// TIA Portal project "正反转流水线控制（核心程序）" (V16)

(* hardware
DEVICE "S7-1200 station_1"  S7-1200 Station
   slot 0: "Rack_0"  S7-1200 Rack  Rack  V1.0
   slot 1: "PLC_1"  CPU 1214C DC/DC/Rly  6ES7 214-1HG40-0XB0  V4.4
DEVICE "HMI_1"  KTP700 Basic PN
   slot 0: "HMI_1"  KTP700 Basic PN  6AV2 123-2GB03-0AX0  16.0.0.0
   slot 1: "HMI_RT_1"  KTP700 Basic PN  6AV2 123-2GB03-0AX0  16.0.0.0
   slot 5: "HMI_1.IE_CP_1"  PROFINET Interface  16.0.0.0
      slot 1: "PROFINET Interface_1"  PROFINET Interface
         slot 1: "Port_1"  Port
*)

// ===== PLC "PLC_1"  CPU 1214C DC/DC/Rly =====

VAR_GLOBAL   // PLC tag table "默认变量表"
   "Tag_1" AT %M20.0 : Bool;
END_VAR

VAR_GLOBAL   // PLC tag table "中间变量"
   "启动(1)" AT %M0.0 : Bool;
   "停止" AT %M0.1 : Bool;
   "复位(1)" AT %M0.2 : Bool;
   "启动标志" AT %M0.3 : Bool;
   "中间寄存器1" AT %MD100 : DInt;
   "收料皮带启动" AT %M0.4 : Bool;
   "中间寄存器2" AT %MD104 : DInt;
   "判断是否" AT %M0.5 : Bool;
   "中间变量1" AT %M0.6 : Bool;
   "中间寄存器3" AT %MD108 : DInt;
   "中间变量2" AT %M0.7 : Bool;
   "中间变量2(1)" AT %M1.0 : Bool;
   "中间变量3" AT %M1.1 : Bool;
END_VAR

VAR_GLOBAL   // PLC tag table "io表"
   "上料端传感器" AT %I2.0 : Bool;
   "中断传感器" AT %I2.1 : Bool;
   "下料传感器" AT %I2.2 : Bool;
   "启动" AT %I2.3 : Bool;
   "复位" AT %I2.4 : Bool;
   "急停" AT %I2.5 : Bool;
   "挡位1" AT %I2.6 : Bool;
   "急停按钮" AT %I2.7 : Bool;
   "FACTORY I/O (Running)" AT %I1.0 : Bool;
   "卡槽" AT %Q2.0 : Bool;
   "绿色" AT %Q2.1 : Bool;
   "黄色" AT %Q2.2 : Bool;
   "红色" AT %Q2.3 : Bool;
   "上料" AT %Q2.4 : Bool;
   "取料" AT %Q2.5 : Bool;
   "速度" AT %ID30 : Real;
   "皮带1" AT %QD30 : Real;
   "皮带2" AT %QD34 : Real;
   "显示屏" AT %QD38 : DInt;
END_VAR

DATA_BLOCK "数据块_1"   // DB1
{ S7_Optimized_Access := 'TRUE' }
VERSION : 0.1
   VAR
      中间变量1 : Bool := 0;
      中间变量2 : Bool := 0;
   END_VAR
BEGIN
END_DATA_BLOCK

FUNCTION "MHJ-PLC-Lab-Function-S71200" : Void   // FC9000, SCL
{ S7_Optimized_Access := 'TRUE' }
VERSION : 0.1
   VAR_TEMP
      rdTimeReturn : Int;
      outputTime : DTL;
      SyncVal : Byte;
      forVal : Int;
      forVal_2 : Int;
      Value : Byte;
   END_VAR
   VAR CONSTANT
      CompVal : Byte := 16#34;
      Value_01 : Byte := 16#11;
      Value_01_DW : DWord := 16#A165_D992;
      Value_02_DW : DWord := 16#58BE_4401;
   END_VAR
BEGIN

   #Value:=PEEK(area := 16#82,
        dbNumber := 0,
        byteOffset := 511);
   #Value := #Value + 1;

   POKE(area := 16#82,
        dbNumber := 0,
        byteOffset := 511,
        value := #Value);

   POKE(area:=16#81,
        dbNumber:=0,
        byteOffset:=1016,
        value:=#Value_01_DW);
   POKE(area := 16#81,
        dbNumber := 0,
        byteOffset := 1020,
        value := #Value_02_DW);

   POKE(area := 16#81,
        dbNumber := 0,
        byteOffset := 511,
        value := B#16#00);

   FOR #forVal := 0 TO 120 DO
       FOR #forVal_2:=0 TO 10 DO
           #rdTimeReturn:=RD_SYS_T(#outputTime);
           #rdTimeReturn := WR_SYS_T(#outputTime);
           #rdTimeReturn := RD_SYS_T(#outputTime);
           #rdTimeReturn := WR_SYS_T(#outputTime);
       END_FOR;
       #SyncVal:= PEEK(area := 16#81,
                      dbNumber := 0,
                      byteOffset := 511);
       IF #SyncVal = #CompVal THEN
          GOTO M_1;
       END_IF;
   END_FOR;
   RETURN;

   M_1:
   POKE(area := 16#81,
        dbNumber := 0,
        byteOffset := 511,
        value := B#16#0);
END_FUNCTION

ORGANIZATION_BLOCK "Main"   // OB1, LAD, ProgramCycle
TITLE = "Main Program Sweep (Cycle)"
{ S7_Optimized_Access := 'TRUE' }
VERSION : 0.1
   VAR_INPUT
      Initial_Call : Bool;   // Initial call of this OB
      Remanence : Bool;   // =True, if remanent data are available
   END_VAR
   VAR_TEMP   // added for the SCL form of the ladder/FBD networks
      _w1 : Bool;
      _w2 : Bool;
   END_VAR
BEGIN

REGION Network 1
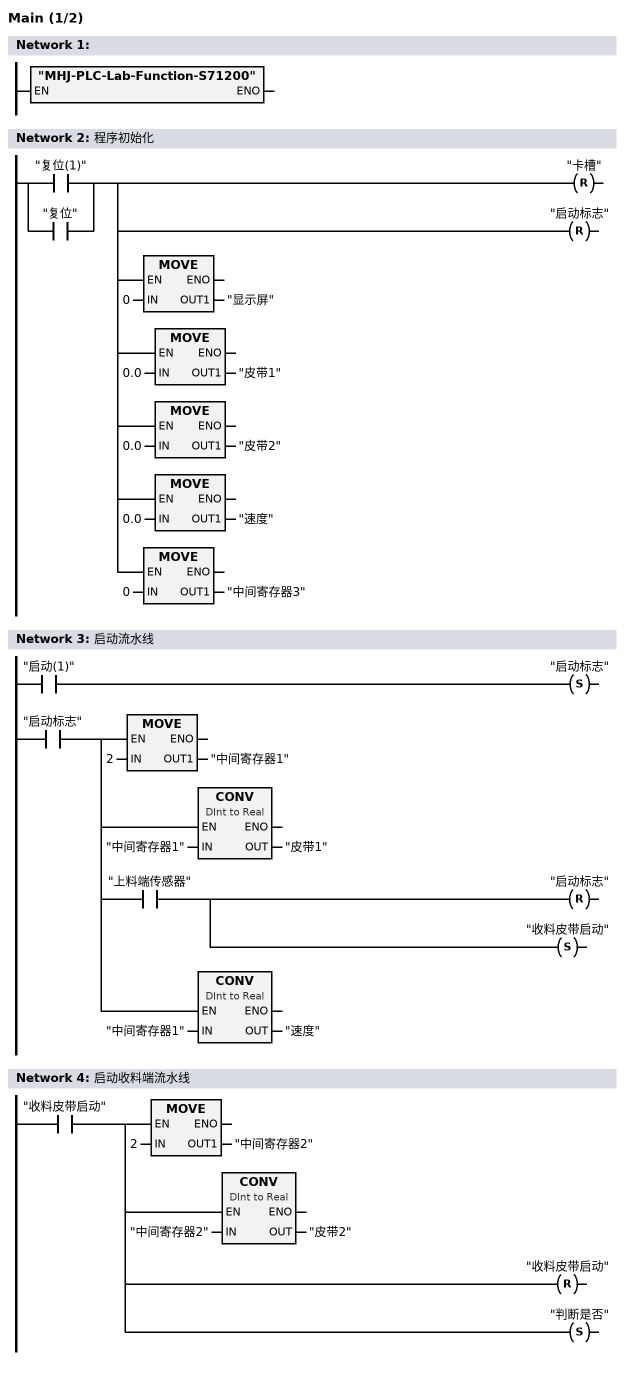
   RUNG wire#powerrail
      "MHJ-PLC-Lab-Function-S71200"()
   END_RUNG
   // the same network as SCL:
   "MHJ-PLC-Lab-Function-S71200"();
END_REGION

REGION Network 2: 程序初始化
   RUNG wire#powerrail
      Contact( "复位(1)" )
      wire#w1
      R_Coil( "卡槽" )
   END_RUNG
   RUNG wire#powerrail
      Contact( "复位" )
   END_RUNG wire#w1
   RUNG wire#w1
      R_Coil( "启动标志" )
   END_RUNG
   RUNG wire#w1
      Move(in := 0, out1 => "显示屏")
   END_RUNG
   RUNG wire#w1
      Move(in := 0.0, out1 => "皮带1")
   END_RUNG
   RUNG wire#w1
      Move(in := 0.0, out1 => "皮带2")
   END_RUNG
   RUNG wire#w1
      Move(in := 0.0, out1 => "速度")
   END_RUNG
   RUNG wire#w1
      Move(in := 0, out1 => "中间寄存器3")
   END_RUNG
   // the same network as SCL:
   IF "复位(1)" OR "复位" THEN
       "卡槽" := FALSE;
       "启动标志" := FALSE;
       "显示屏" := 0;
       "皮带1" := 0.0;
       "皮带2" := 0.0;
       "速度" := 0.0;
       "中间寄存器3" := 0;
   END_IF;
END_REGION

REGION Network 3: 启动流水线
   RUNG wire#powerrail
      Contact( "启动(1)" )
      S_Coil( "启动标志" )
   END_RUNG
   RUNG wire#powerrail
      Contact( "启动标志" )
      wire#w1
      Move(in := 2, out1 => "中间寄存器1")
   END_RUNG
   RUNG wire#w1
      { S7_Templates := "[SrcType := DInt, DestType := Real]" } Convert(in := "中间寄存器1", out => "皮带1")
   END_RUNG
   RUNG wire#w1
      Contact( "上料端传感器" )
      wire#w2
      R_Coil( "启动标志" )
   END_RUNG
   RUNG wire#w2
      S_Coil( "收料皮带启动" )
   END_RUNG
   RUNG wire#w1
      { S7_Templates := "[SrcType := DInt, DestType := Real]" } Convert(in := "中间寄存器1", out => "速度")
   END_RUNG
   // the same network as SCL:
   IF "启动(1)" THEN "启动标志" := TRUE; END_IF;
   IF "启动标志" THEN
       "中间寄存器1" := 2;
       "皮带1" := DINT_TO_REAL("中间寄存器1");
   END_IF;
   #_w1 := "启动标志";
   #_w2 := "启动标志" AND "上料端传感器";
   IF #_w2 THEN
       "启动标志" := FALSE;
       "收料皮带启动" := TRUE;
   END_IF;
   IF #_w1 THEN "速度" := DINT_TO_REAL("中间寄存器1"); END_IF;
END_REGION

REGION Network 4: 启动收料端流水线
   RUNG wire#powerrail
      Contact( "收料皮带启动" )
      wire#w1
      Move(in := 2, out1 => "中间寄存器2")
   END_RUNG
   RUNG wire#w1
      { S7_Templates := "[SrcType := DInt, DestType := Real]" } Convert(in := "中间寄存器2", out => "皮带2")
   END_RUNG
   RUNG wire#w1
      R_Coil( "收料皮带启动" )
   END_RUNG
   RUNG wire#w1
      S_Coil( "判断是否" )
   END_RUNG
   // the same network as SCL:
   IF "收料皮带启动" THEN
       "中间寄存器2" := 2;
       "皮带2" := DINT_TO_REAL("中间寄存器2");
   END_IF;
   #_w1 := "收料皮带启动";
   IF #_w1 THEN
       "收料皮带启动" := FALSE;
       "判断是否" := TRUE;
   END_IF;
END_REGION

REGION Network 5: 计数
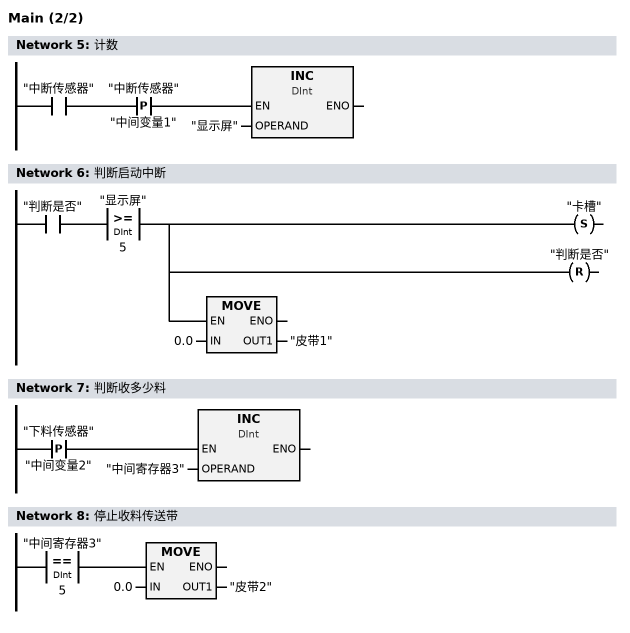
   RUNG wire#powerrail
      Contact( "中断传感器" )
      P_Contact(operand := "中断传感器", bit := "中间变量1")
      { S7_Templates := "DestType := DInt" } Inc( "显示屏" )
   END_RUNG
   // the same network as SCL:
   #_w1 := "中断传感器" AND "中断传感器" AND NOT "中间变量1";   // rising edge of "中断传感器"
   "中间变量1" := "中断传感器";
   IF #_w1 THEN "显示屏" := "显示屏" + 1; END_IF;
END_REGION

REGION Network 6: 判断启动中断
   RUNG wire#powerrail
      Contact( "判断是否" )
      { S7_Templates := "SrcType := DInt" } GE_Contact(in1 := "显示屏", in2 := 5)
      wire#w1
      S_Coil( "卡槽" )
   END_RUNG
   RUNG wire#w1
      R_Coil( "判断是否" )
   END_RUNG
   RUNG wire#w1
      Move(in := 0.0, out1 => "皮带1")
   END_RUNG
   // the same network as SCL:
   IF "判断是否" AND ("显示屏" >= 5) THEN "卡槽" := TRUE; END_IF;
   #_w1 := "判断是否" AND ("显示屏" >= 5);
   IF #_w1 THEN
       "判断是否" := FALSE;
       "皮带1" := 0.0;
   END_IF;
END_REGION

REGION Network 7: 判断收多少料
   RUNG wire#powerrail
      P_Contact(operand := "下料传感器", bit := "中间变量2")
      { S7_Templates := "DestType := DInt" } Inc( "中间寄存器3" )
   END_RUNG
   // the same network as SCL:
   #_w1 := "下料传感器" AND NOT "中间变量2";   // rising edge of "下料传感器"
   "中间变量2" := "下料传感器";
   IF #_w1 THEN "中间寄存器3" := "中间寄存器3" + 1; END_IF;
END_REGION

REGION Network 8: 停止收料传送带
   RUNG wire#powerrail
      { S7_Templates := "SrcType := DInt" } EQ_Contact(in1 := "中间寄存器3", in2 := 5)
      Move(in := 0.0, out1 => "皮带2")
   END_RUNG
   // the same network as SCL:
   IF "中间寄存器3" = 5 THEN "皮带2" := 0.0; END_IF;
END_REGION
END_ORGANIZATION_BLOCK

(* ===== HMI "HMI_RT_1" =====
system functions are stored by id; their names below are inferred from use
connection "HMI_连接_1": ETHERNET, SMART_S7_1200_OMS

HMI tags "默认变量表"
   "Tag_ScreenNumber" : UInt, internal
   "启动(1)" : Bool = PLC "启动(1)" AT %M0.0, 1 s
   "复位(1)" : Bool = PLC "复位(1)" AT %M0.2, 1 s

Template "模板_1" 800x480
   Button "退出" at 714,429 size 71x50; TextOff '退出'; PictureOff "ExitRuntime_KTP700_Basic_PN_TR"; PictureOn "ExitRuntime_KTP700_Basic_PN_TR"
      on Release: StopRuntime(0)
   Button "Template_Button" at 614,429 size 71x50; TextOff 'Text'
   Button "Template_Button_1" at 514,429 size 71x50; TextOff 'Text'
   Button "Template_Button_2" at 414,429 size 71x50; TextOff 'Text'
   Button "Template_Button_3" at 314,429 size 71x50; TextOff 'Text'
   Button "Template_Button_4" at 214,429 size 71x50; TextOff 'Text'
   Button "Template_Button_5" at 114,429 size 71x50; TextOff 'Text'
   Button "起始画面" at 14,429 size 71x50; TextOff '起始画面'; PictureOff "NavigateHome_KTP700_Basic_PN_TR"; PictureOn "NavigateHome_KTP700_Basic_PN_TR"
      on Release: ActivateScreen("根画面", 0)
   SymbolicIOField "Symbolic_IO_Field_Screen" at 93,9 size 600x33; TextOff '0'; TextOn '1'; TextList "TextList_ScreenNames"
      ProcessValue <- "Tag_ScreenNumber"
      on Change: ActivateScreenByNumber("Tag_ScreenNumber", 0)
   DateTimeField "HmiScreenItemData" at 695,25 size 105x25
   DateTimeField "HmiScreenItemData_1" at 695,0 size 105x25
   GraphicView "Logo" at 0,0 size 91x51; Picture "HMI_1 的 Logo"

screen "根画面" 800x480, template "模板_1"
   on GenerateScreen: SetTag("Tag_ScreenNumber", 1)
   Button "按钮_1" at 206,171 size 96x32; TextOff '启动'
      on Press: SetBit("启动(1)")
      on Release: ResetBit("启动(1)")
   Button "按钮_2" at 207,240 size 96x32; TextOff '复位'
      on Release: ResetBit("复位(1)")
      on Press: SetBit("复位(1)")
*)